INTERFACE ITF_BaseLogger_HMI_Connector_Command

END_INTERFACE

(* stored: Version 1.1.0.1
   Itf ITF_BaseLogger_HMI_Connector_Command: Id {fe1bd24b-1818-07f0-3c99-81114f5ac2d9} *)
